INTERFACE I_NodeFactoryVisitor

METHOD VisitNodeFactory
VAR_INPUT
	VisitingNodeFactory : I_NodePrototypes;
END_VAR
END_METHOD

END_INTERFACE

(* stored: Version 1.1.0.1, ProductVersion 3.1.4024.12
   Itf I_NodeFactoryVisitor: Id {1d8fa654-02cc-02ab-1175-6487c46b7d24}
   Method VisitNodeFactory: Id {cf6a55c0-d0a7-0f61-0fe2-96bf6b707b33} *)
